INTERFACE I_Cylinder

END_INTERFACE

(* stored: Version 1.1.0.1, ProductVersion 3.1.4024.12
   Itf I_Cylinder: Id {19a257a1-962d-488e-a322-9edd1b71d208} *)
